# EPICS IOC start-up script: iocsh/EthercatMCAxishome.iocsh
dbLoadRecords("EthercatMChome.template", "PREFIX=$(PREFIX), MOTOR_NAME=$(MOTOR_NAME), MOTOR_PORT=$(MOTOR_PORT), AXIS_NO=$(AXIS_NO), PREC=3")
